// TIA Portal V18 export
DATA_BLOCK "alm_DB"   // DB37
VERSION : 0.1
// stored: AutoNumber true, DBAccessibleFromOPCUA true, InstanceOfName alm, InstanceOfType FB
"alm"
   // VAR_INPUT
   //    alarm_input : Array[0..95] of Bool;
   // END_VAR
   // VAR_OUTPUT
   //    alarmreg_output : Array[0..95] of Bool;
   // END_VAR
   // VAR_IN_OUT
   //    alarm_ack : Array[0..95] of Bool;
   //    almreset_ons : Bool;
   //    fault_dipslay_reg : Int;
   // END_VAR
   // VAR
   //    i : Int;
   //    alarmregtemp : Array[0..95] of Bool;
   //    temp : Array[0..95] of Bool;
   // END_VAR
BEGIN
END_DATA_BLOCK
